SUBAPPLICATION Uebung_006a3_sub_AX (* Subapplication Type *)
  (* Standard: 61499-2; Description: Copyright (c) 2026 Meisterschulen am Ostbahnhof This program and the accompanying materials are made available under the terms of the Eclipse Public License 2.0 which is available at https://www.eclipse.org/legal/epl-2.0/ SPDX-License-Identifier: EPL-2.0 *)
  (* Version 1.0, 2026-01-13, Moritz Ortmeier, Meisterschulen am Ostbahnhof *)
  PACKAGE Uebungen;
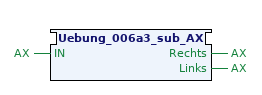
  SOCKETS
    IN : adapter::types::unidirectional::AX;
  END_SOCKETS
  PLUGS
    Rechts : adapter::types::unidirectional::AX;
    Links : adapter::types::unidirectional::AX;
  END_PLUGS
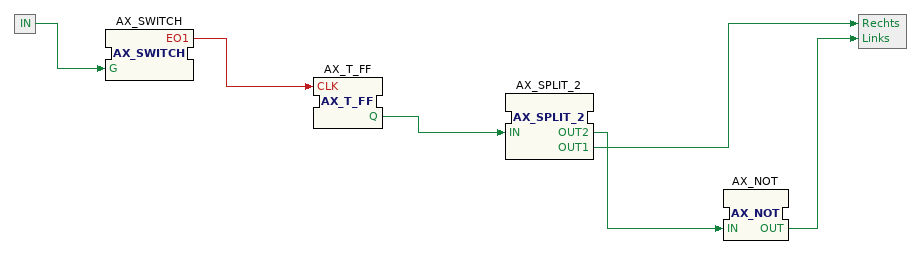
  FBS
    AX_T_FF : adapter::events::unidirectional::AX_T_FF;
    AX_SWITCH : adapter::events::unidirectional::AX_SWITCH;
    AX_NOT : adapter::booleanOperators::AX_NOT;
    AX_SPLIT_2 : adapter::events::unidirectional::AX_SPLIT_2;
  END_FBS
  EVENT_CONNECTIONS
    AX_SWITCH.EO1 TO AX_T_FF.CLK;
  END_CONNECTIONS
  ADAPTER_CONNECTIONS
    IN TO AX_SWITCH.G;
    AX_NOT.OUT TO Links;
    AX_T_FF.Q TO AX_SPLIT_2.IN;
    AX_SPLIT_2.OUT2 TO AX_NOT.IN;
    AX_SPLIT_2.OUT1 TO Rechts;
  END_CONNECTIONS
END_SUBAPPLICATION
